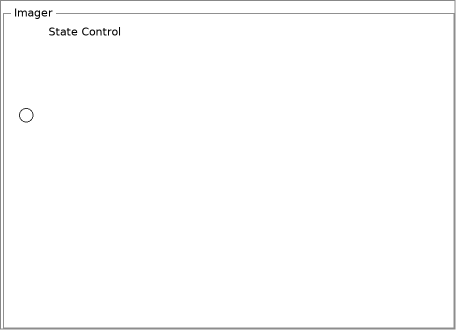
VISUALIZATION ImagerGUI  // 456x330
VAR_IN_OUT
	fbDev	:	FB_ExampleDevice;
END_VAR
    GroupBox (3,5 451x323), "Imager"
        RadioButton (14,49 97x122), variable: fbDev.stDevice.nRequestedState
            Areas[1]: Text=State 1
            Areas[2]: Text=State 2
            Areas[3]: Text=State 3
        Label (7,12 150x30), "State Control"
END_VISUALIZATION

(* stored: Version 1.1.0.1, ProductVersion 3.1.4022.12
   Visu ImagerGUI: Id {c4e9eed9-0847-0b0c-1a64-5b138d22d3b0} *)
